TYPE ST_EventClassInfo :
STRUCT
	GUID : GUID;
	BaseAddress : POINTER TO TcEventEntry;
	Count : UDINT;
END_STRUCT
END_TYPE

(* stored: Version 1.1.0.1, ProductVersion 3.1.4024.12
   DUT ST_EventClassInfo: Id {487a2889-ffa0-4e42-9beb-25bf846e8ad6} *)
